INTERFACE IDrive

METHOD MoveAbsolute : TcoCore.ITcoTaskStatus
VAR_INPUT
	TargetPosition : LREAL;
END_VAR
END_METHOD

END_INTERFACE

(* stored: Version 1.1.0.1, ProductVersion 3.1.4024.6
   Itf IDrive: Id {56a4a9b0-da64-4b93-9928-f728021459b0}
   Method MoveAbsolute: Id {c317d00a-5ad5-412f-88c4-709bf3587e00} *)
